// Brief: Master Arm Initialization
FUNCTION_BLOCK PUBLIC FB_ArmCart EXTENDS FB_MasterArmCtrlBase
VAR_INPUT
END_VAR
VAR_OUTPUT
END_VAR
VAR
END_VAR

END_FUNCTION_BLOCK

(* stored: Version 1.1.0.1, ProductVersion 3.1.4024.12
   POU FB_ArmCart: Id {acf69b98-a94c-45d6-930a-e719a9a02026}, SpecialFunc None *)
